# EPICS autosave request: iocBoot/ioc13LAE500/auto_settings.req
file "Newport_LAE500_settings.req",     P=13LAE500:, R=LAE500
file "scan_settings.req",               P=13LAE500:, S=scan1
file "scan_settings.req",               P=13LAE500:, S=scan2
file "scan_settings.req",               P=13LAE500:, S=scan3
file "scan_settings.req",               P=13LAE500:, S=scan4
